// TIA Portal V20 export
TYPE "LBP_typeNCKProcessIRTFlags"
TITLE = LBP_NCKProcessIRT Output Interface / LBP_NCKProcessIRT Interface sortie
// User data type for LBP_NCKProcessIRT[FC3] Output Parameters / Type de données utilisateur pour LBP_NCKProcessIRT[FC3] Paramètres de sortie
   STRUCT
      IRFromNck : Bool;   // Interrupt from NCK / Interruption en provenance du NCK
      TM : Bool;   // Tool change / Changement d'outil
      InPosition : Array[1..31] of Bool;   // Axis or spindle position reached / Position d'axe ou de broche atteinte
      AuxFunction : Array[1..10] of Bool;   // Auxiliary function available / Fonction auxiliaire disponible
   END_STRUCT;
END_TYPE
